Fanuc KAREL source: kx00014.KL

-- PROVISIONAL review KL for V1013-1; original PC SHA256 9232e09443f017920e7372e4938919b5fc001d3b8e2b049f9392f14a293e65e1
-- Incomplete behavior may be omitted. Consult companion uncertainty JSON. Do not deploy.
PROGRAM KX00014
%NOLOCKGROUP
VAR
  I : INTEGER
  J : INTEGER
  B : BOOLEAN
  F : FILE
  S : STRING[80]
-- UNRESOLVED_DECL P type=000102
BEGIN
  -- UNRESOLVED_PC offsets 5-7; opcodes 9D,3C
  -- UNRESOLVED_PC offsets 12-16; opcodes 7F
END KX00014
